{attribute 'GeneratedUsingTerminal: BK1120-0000-0016'}
{attribute addProperty BoxType "BK1120-0000-0016"}
{attribute addProperty Id "Term_376_KL1002KL1002_BB38DA8F0"}
{attribute addProperty CRC "2365677117"}
{attribute addProperty Size "0"}
TYPE A_0003_BK1120_0000_0016_8D015E3D EXTENDS BK1120_AEEC0900 :
STRUCT
	{attribute addProperty Name "Term_376_KL1002"}
	Term_376_KL1002 : KL1002_BB38DA8F;
END_STRUCT
END_TYPE

(* stored: Version 1.2.0.0, ProductVersion 3.1.4024.9
   DUT A_0003_BK1120_0000_0016_8D015E3D: Id {327e9694-7a10-41cb-8caf-7970b941929c} *)
